// TIA Portal V18 export
FUNCTION_BLOCK "ER_HMI_btnColor"   // FB2, FBD
{ S7_Optimized_Access := 'TRUE' }
VERSION : 0.1
// stored: AutoNumber true, IsIECCheckEnabled false, IsRetainMemResEnabled false, MemoryReserve 100, SetENOAutomatically false, UDAEnableTagReadback false
   VAR_INPUT
      xER : Bool;
      xWN : Bool;
   END_VAR
   VAR_OUTPUT
      color : Int;
   END_VAR
   VAR CONSTANT
      c0clear : Int := 0;
      c1alarm : Int := 1;
      c2warning : Int := 2;
   END_VAR
BEGIN

REGION Network 1 (SCL)
   IF #xER THEN
       #color := #c1alarm;
   ELSIF #xWN THEN
       #color := #c2warning;
   ELSE
       #color := #c0clear;
   END_IF;
END_REGION
END_FUNCTION_BLOCK
